Staubli VAL3: JOINT.dtx

public num distance
public num moveType
public num nIndexGun
public num nTime
public num nStop
public num nTcpAction
public num nFrameIndex
public num nGasPressure
public num nLaserPower
public num nPWMPercent
public num nJointMode
public string comment
public string instruction
public bool toStop
public frame fTrack = {fatherId=world[0]}
public jointRx jJoints
public mdesc nom_speed = {vel=30, tmax=9999, rmax=9999, leave=30, reach=30}
